KUKA KRL data list: $config.dat

&ACCESS RVO1
&COMMENT
DEFDAT $config PUBLIC

DECL BOOL KUSTIC_START
DECL BOOL KUSTIC_STOP
DECL BOOL KUSTIC_PLAYING_STATUS
DECL BOOL KUSTIC_EMERGENCY
DECL BOOL KUSTIC_CALIBRATE

STRUC KUSTIC_STRUC FRAME POINT, INT TEMPO

DECL KUSTIC_STRUC POINTS[30]

ENDDAT
